Staubli VAL3: Language.pgx

program Language()
  local num l_nKey
begin
  userPage()
  cls()
  call xyPut(5,3,"Please Choose Your Language")
  call xyPut(5,5,"F1. Chinese")
  call xyPut(5,6,"F2. English")


  // while true
  //   l_nKey=getKey()
  //  switch l_nKey
  //    case 271
  //      sLanguge="Chinese"
  //      return
  //    break
  //    case 272
  //      sLanguge="English"
  //      return
  //    break
  //  endSwitch
  //delay(0)
  //endWhile
  sLanguge="Chinese"
end
